PROGRAM System
VAR
	ElectricBoard: ElectricBoard;
	ConveyorEntry: ConveyorEntry;
	TransferConveyor: TransferConveyor;
	TransferToLeftorRight: TransferToLeftorRight;
END_VAR

//System functions.
ElectricBoard();
ConveyorEntry();
TransferConveyor();
TransferToLeftorRight();

END_PROGRAM

(* stored: Version 1.1.0.1, ProductVersion 3.1.4024.6
   POU System: Id {d7288777-637e-42ff-af45-8ccee0e2f8c6}, SpecialFunc None *)
